(* Logix 5000 project; controller Lavado Emulate 5570 rev 32.11; software revision 32.00 *)
// Lavadora de botellas simplificada; ciclo automatico continuo basado en GRAFCET Nivel 3 v02 y CR-001; cambio CR-002.

TASK MainTask (continuous, watchdog 500 ms) : P_Lavadora

MODULES
   Local : Emulate 5570 (ICP 2, rev 32.11)
END_MODULES

VAR_GLOBAL   (* controller tags *)
   ACT_LAV_Alineacion : BOOL;   // Salida NX: 1 extiende alineador; 0 retrae.
   ACT_LAV_Banda : BOOL;   // Salida NX: 1 mueve banda; 0 detiene.
   ACT_LAV_CierrePinzas : BOOL;   // Salida NX: 1 cierra pinzas; 0 abre.
   ACT_LAV_Detencion : BOOL;   // Salida NX: 0 retiene; 1 libera.
   ACT_LAV_DetencionEntrada : BOOL;   // Salida NX CR-001: 1 extiende; 0 retrae.
   ACT_LAV_GiroLavado : BOOL;   // Salida NX: 1 gira a lavado; 0 retorna a origen.
   CMD_Inicio : BOOL;   // Pulso de inicio del automatico continuo.
   CMD_Parada : BOOL;   // Pulso de parada; cancela el lote y ordena posiciones iniciales.
   CMD_Reinicio : BOOL;   // Pulso de reinicio; borra etapas, contadores y temporizadores y ordena posiciones iniciales.
   SE_LAV_Alineado : BOOL;   // Entrada NX: alineador extendido.
   SE_LAV_CierrePinza : BOOL;   // Entrada NX: pinzas cerradas.
   SE_LAV_ConteoSalida : BOOL;   // Entrada NX: sensor de salida; cuenta por flanco ascendente.
   SE_LAV_DetencionEntradaExtendido : BOOL;   // Entrada NX CR-001: detencion de entrada extendida.
   SE_LAV_DetencionEntradaRetraido : BOOL := 1;   // Entrada NX CR-001: detencion de entrada retraida.
   SE_LAV_EntradaBotellas : BOOL;   // Entrada NX: sensor de entrada; cuenta por flanco ascendente.
   SE_LAV_Giro : BOOL;   // Entrada NX: giro en posicion de lavado.
   SE_LAV_SinAlinear : BOOL := 1;   // Entrada NX: alineador retraido.
   SE_LAV_SinDetencion : BOOL;   // Entrada NX: brazo de salida retirado y paso libre.
   SE_LAV_SinGiro : BOOL := 1;   // Entrada NX: giro en origen.
   T_Cierre : TIMER := (PRE := 1000);
END_VAR

PROGRAM P_Lavadora   (* main routine R00_Main *)
// Control secuencial simplificado; tres mandos, dos contadores, dos temporizadores y ciclo continuo.
VAR
   C_EntradaLote : COUNTER := (PRE := 7);   // Cuenta siete botellas de entrada por flanco ascendente.
   C_SalidaLote : COUNTER := (PRE := 7);   // Cuenta siete botellas de salida por flanco ascendente.
   MEM_ONS_ConteoSalida : BOOL;   // Memoria ONS exclusiva del sensor de salida.
   MEM_ONS_EntradaBotellas : BOOL;   // Memoria ONS exclusiva del sensor de entrada.
   MEM_ONS_Inicio : BOOL;   // Memoria ONS exclusiva de CMD_Inicio.
   MEM_ONS_Parada : BOOL;   // Memoria ONS exclusiva de CMD_Parada.
   MEM_ONS_Reinicio : BOOL;   // Memoria ONS exclusiva de CMD_Reinicio.
   PUL_EntradaBotella : BOOL;   // Pulso de un scan por botella de entrada.
   PUL_Inicio : BOOL;   // Pulso de un scan para inicio.
   PUL_Parada : BOOL;   // Pulso de un scan para parada.
   PUL_Reinicio : BOOL;   // Pulso de un scan para reinicio.
   PUL_SalidaBotella : BOOL;   // Pulso de un scan por botella de salida.
   ST_CicloAutomatico : BOOL;   // Memoria de marcha del ciclo automatico continuo.
   ST_LoteEntradaCompleto : BOOL;   // Memoria del septimo flanco de entrada antes del RES.
   ST_LoteSalidaCompleto : BOOL;   // Memoria del septimo flanco de salida antes del RES.
   T_Asentamiento : TIMER := (PRE := 2500);   // Ajuste de posicion de botellas despues de extender la detencion de entrada.
   T_Lavado : TIMER := (PRE := 3000);   // Tiempo de lavado del lote.
   T_Lavado_pos : TIMER := (PRE := 1000);
   TR_T00 : BOOL;   // Transicion de espera a alimentacion.
   TR_T10 : BOOL;   // Transicion despues de siete entradas.
   TR_T100 : BOOL;   // Transicion despues de siete salidas.
   TR_T105 : BOOL;   // Transicion con fin de lote seguro.
   TR_T110 : BOOL;   // Transicion automatica al siguiente lote.
   TR_T12 : BOOL;   // Transicion con detencion de entrada extendida.
   TR_T15 : BOOL;   // Transicion al completar posicionamiento.
   TR_T20 : BOOL;   // Transicion con alineador extendido.
   TR_T30 : BOOL;   // Transicion con pinzas cerradas.
   TR_T40 : BOOL;   // Transicion con giro en lavado.
   TR_T50 : BOOL;   // Transicion al completar tiempo de lavado.
   TR_T60 : BOOL;   // Transicion con giro en origen.
   TR_T70 : BOOL;   // Transicion con pinzas abiertas.
   TR_T80 : BOOL;   // Transicion con alineador retraido.
   TR_T90 : BOOL;   // Transicion con salida liberada.
   X00_Inicial : BOOL := 1;   // Etapa 0: espera de inicio y posiciones iniciales.
   X100_EvacuandoLote : BOOL;   // Etapa 100: evacuar y contar salidas.
   X105_CerrandoSalidaFinLote : BOOL;   // Etapa 105: cerrar salida y confirmar fin seguro.
   X10_Alimentando : BOOL;   // Etapa 10: alimentar y contar entradas.
   X110_RetraiendoDetencionEntrada : BOOL;   // Etapa 110: retraer detencion de entrada.
   X12_ExtendiendoDetencionEntrada : BOOL;   // Etapa 12: extender detencion de entrada con banda activa.
   X15_Posicionando : BOOL;   // Etapa 15: acomodar lote con banda activa.
   X20_Alineando : BOOL;   // Etapa 20: extender alineador.
   X30_CerrandoPinzas : BOOL;   // Etapa 30: cerrar pinzas.
   X40_GirandoLavado : BOOL;   // Etapa 40: girar hacia lavado.
   X50_Lavando : BOOL;   // Etapa 50: mantener lavado temporizado.
   X60_RegresandoGiro : BOOL;   // Etapa 60: regresar giro al origen.
   X70_AbriendoPinzas : BOOL;   // Etapa 70: abrir pinzas.
   X80_RetirandoAlineador : BOOL;   // Etapa 80: retraer alineador.
   X90_DesbloqueandoSalida : BOOL;   // Etapa 90: liberar salida.
END_VAR

ROUTINE R00_Main   (* ladder *)
// Despacha seis rutinas en orden determinista de scan.
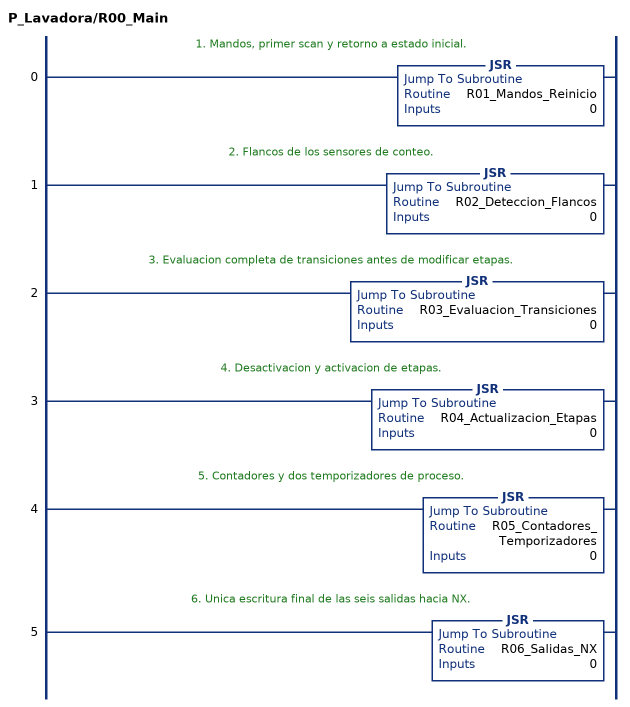
   // 1. Mandos, primer scan y retorno a estado inicial.
   0: JSR(R01_Mandos_Reinicio,0);
   // 2. Flancos de los sensores de conteo.
   1: JSR(R02_Deteccion_Flancos,0);
   // 3. Evaluacion completa de transiciones antes de modificar etapas.
   2: JSR(R03_Evaluacion_Transiciones,0);
   // 4. Desactivacion y activacion de etapas.
   3: JSR(R04_Actualizacion_Etapas,0);
   // 5. Contadores y dos temporizadores de proceso.
   4: JSR(R05_Contadores_Temporizadores,0);
   // 6. Unica escritura final de las seis salidas hacia NX.
   5: JSR(R06_Salidas_NX,0);
END_ROUTINE

ROUTINE R01_Mandos_Reinicio   (* ladder *)
// Tres mandos: inicio, parada y reinicio; parada/reinicio ordenan estado inicial.
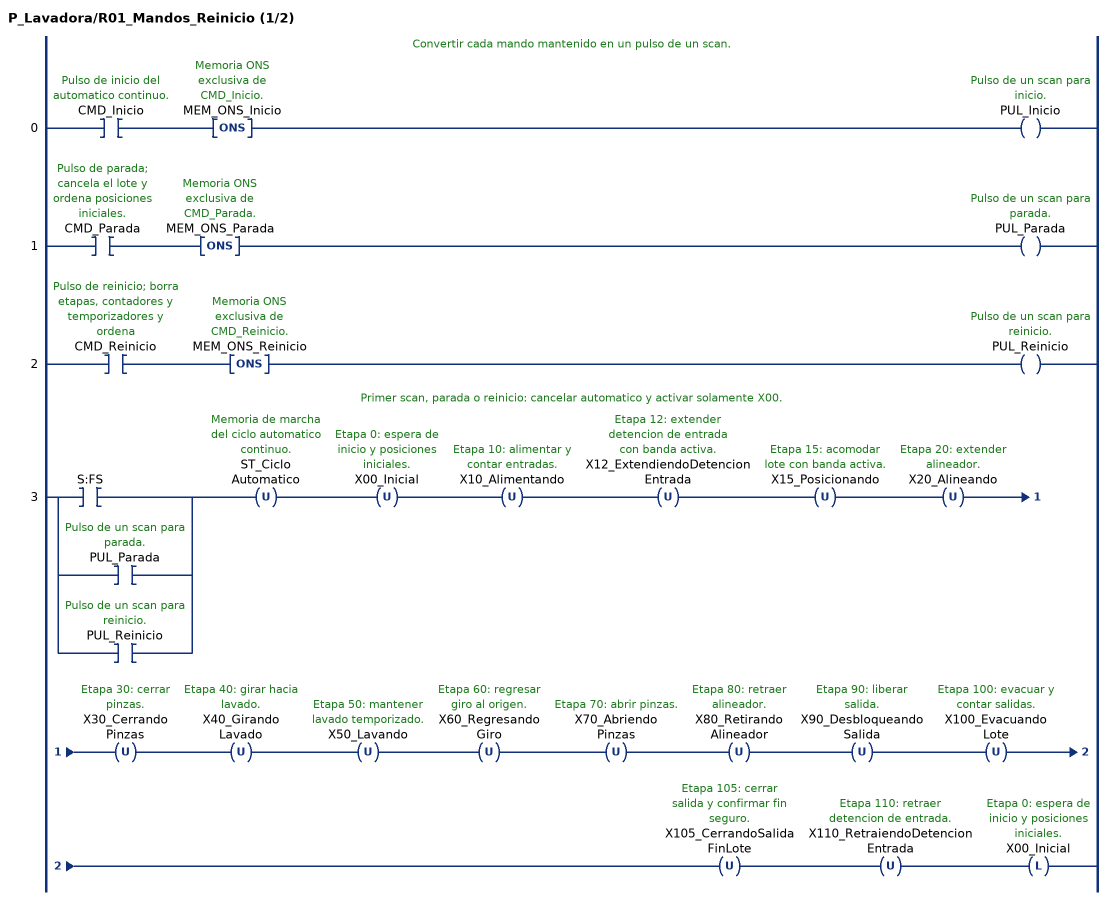
   // Convertir cada mando mantenido en un pulso de un scan.
   0: XIC(CMD_Inicio)ONS(MEM_ONS_Inicio)OTE(PUL_Inicio);
   1: XIC(CMD_Parada)ONS(MEM_ONS_Parada)OTE(PUL_Parada);
   2: XIC(CMD_Reinicio)ONS(MEM_ONS_Reinicio)OTE(PUL_Reinicio);
   // Primer scan, parada o reinicio: cancelar automatico y activar solamente X00.
   3: [XIC(S:FS) ,XIC(PUL_Parada) ,XIC(PUL_Reinicio) ]OTU(ST_CicloAutomatico)OTU(X00_Inicial)OTU(X10_Alimentando)OTU(X12_ExtendiendoDetencionEntrada)OTU(X15_Posicionando)OTU(X20_Alineando)OTU(X30_CerrandoPinzas)OTU(X40_GirandoLavado)OTU(X50_Lavando)OTU(X60_RegresandoGiro)OTU(X70_AbriendoPinzas)OTU(X80_RetirandoAlineador)OTU(X90_DesbloqueandoSalida)OTU(X100_EvacuandoLote)OTU(X105_CerrandoSalidaFinLote)OTU(X110_RetraiendoDetencionEntrada)OTL(X00_Inicial);
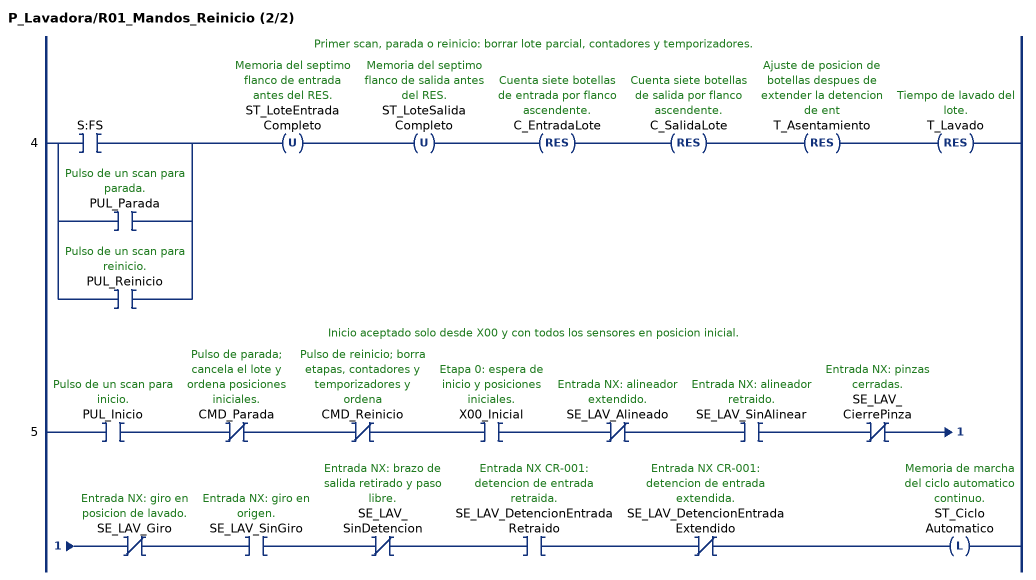
   // Primer scan, parada o reinicio: borrar lote parcial, contadores y temporizadores.
   4: [XIC(S:FS) ,XIC(PUL_Parada) ,XIC(PUL_Reinicio) ]OTU(ST_LoteEntradaCompleto)OTU(ST_LoteSalidaCompleto)RES(C_EntradaLote)RES(C_SalidaLote)RES(T_Asentamiento)RES(T_Lavado);
   // Inicio aceptado solo desde X00 y con todos los sensores en posicion inicial.
   5: XIC(PUL_Inicio)XIO(CMD_Parada)XIO(CMD_Reinicio)XIC(X00_Inicial)XIO(SE_LAV_Alineado)XIC(SE_LAV_SinAlinear)XIO(SE_LAV_CierrePinza)XIO(SE_LAV_Giro)XIC(SE_LAV_SinGiro)XIO(SE_LAV_SinDetencion)XIC(SE_LAV_DetencionEntradaRetraido)XIO(SE_LAV_DetencionEntradaExtendido)OTL(ST_CicloAutomatico);
END_ROUTINE

ROUTINE R02_Deteccion_Flancos   (* ladder *)
// Cuenta una vez cada botella aunque el sensor permanezca activo.
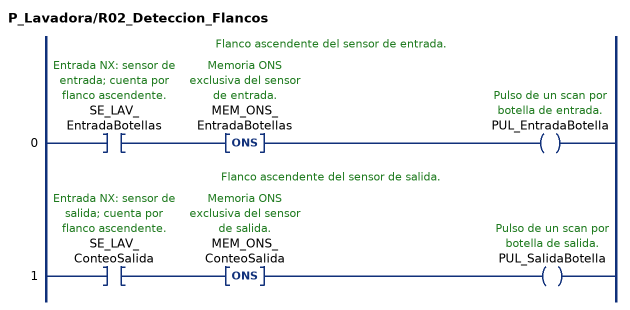
   // Flanco ascendente del sensor de entrada.
   0: XIC(SE_LAV_EntradaBotellas)ONS(MEM_ONS_EntradaBotellas)OTE(PUL_EntradaBotella);
   // Flanco ascendente del sensor de salida.
   1: XIC(SE_LAV_ConteoSalida)ONS(MEM_ONS_ConteoSalida)OTE(PUL_SalidaBotella);
END_ROUTINE

ROUTINE R03_Evaluacion_Transiciones   (* ladder *)
// Evalua las quince transiciones del GRAFCET sin modificar etapas.
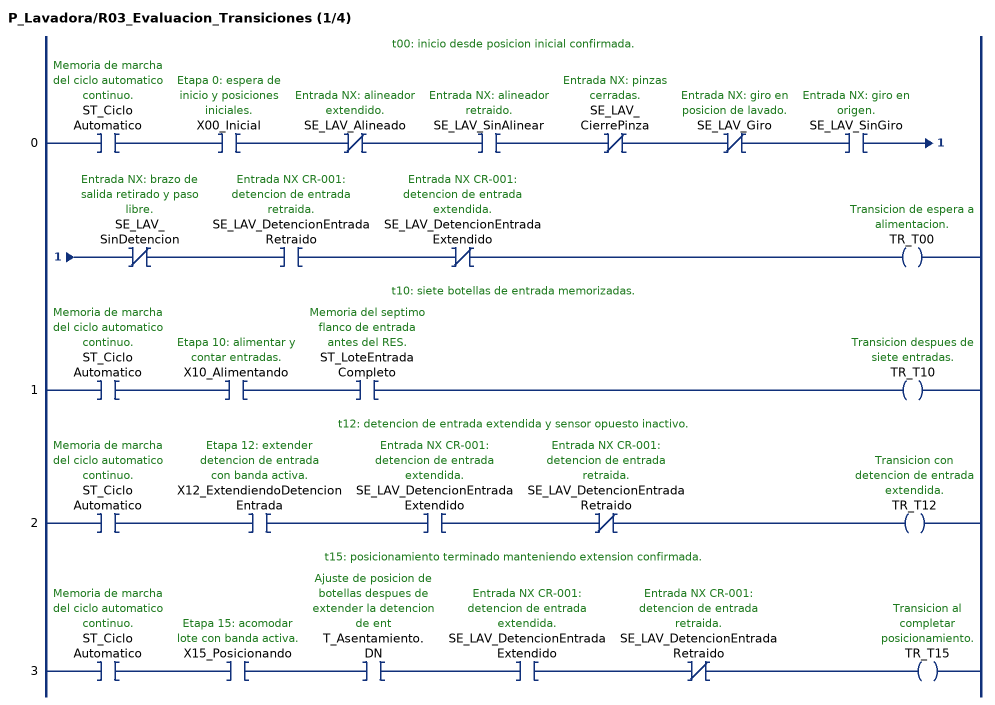
   // t00: inicio desde posicion inicial confirmada.
   0: XIC(ST_CicloAutomatico)XIC(X00_Inicial)XIO(SE_LAV_Alineado)XIC(SE_LAV_SinAlinear)XIO(SE_LAV_CierrePinza)XIO(SE_LAV_Giro)XIC(SE_LAV_SinGiro)XIO(SE_LAV_SinDetencion)XIC(SE_LAV_DetencionEntradaRetraido)XIO(SE_LAV_DetencionEntradaExtendido)OTE(TR_T00);
   // t10: siete botellas de entrada memorizadas.
   1: XIC(ST_CicloAutomatico)XIC(X10_Alimentando)XIC(ST_LoteEntradaCompleto)OTE(TR_T10);
   // t12: detencion de entrada extendida y sensor opuesto inactivo.
   2: XIC(ST_CicloAutomatico)XIC(X12_ExtendiendoDetencionEntrada)XIC(SE_LAV_DetencionEntradaExtendido)XIO(SE_LAV_DetencionEntradaRetraido)OTE(TR_T12);
   // t15: posicionamiento terminado manteniendo extension confirmada.
   3: XIC(ST_CicloAutomatico)XIC(X15_Posicionando)XIC(T_Asentamiento.DN)XIC(SE_LAV_DetencionEntradaExtendido)XIO(SE_LAV_DetencionEntradaRetraido)OTE(TR_T15);
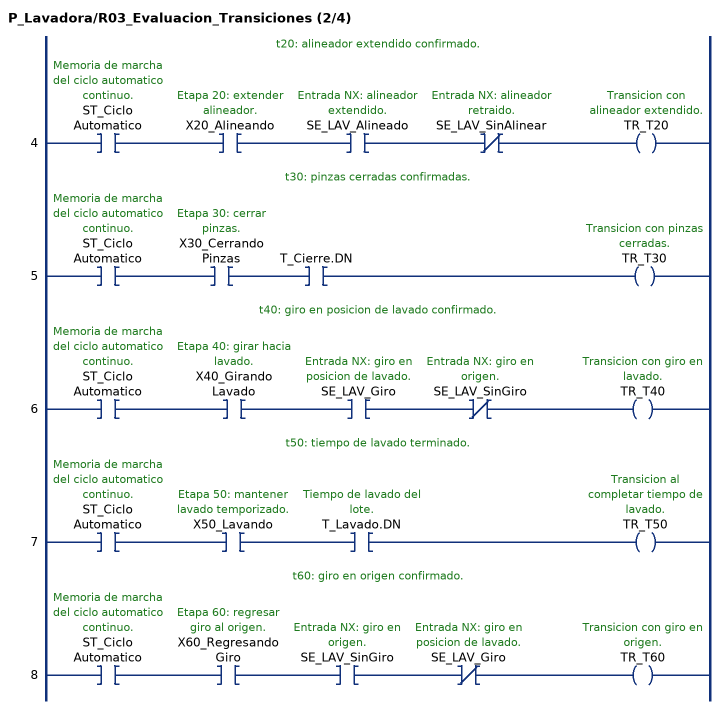
   // t20: alineador extendido confirmado.
   4: XIC(ST_CicloAutomatico)XIC(X20_Alineando)XIC(SE_LAV_Alineado)XIO(SE_LAV_SinAlinear)OTE(TR_T20);
   // t30: pinzas cerradas confirmadas.
   5: XIC(ST_CicloAutomatico)XIC(X30_CerrandoPinzas)XIC(T_Cierre.DN)OTE(TR_T30);
   // t40: giro en posicion de lavado confirmado.
   6: XIC(ST_CicloAutomatico)XIC(X40_GirandoLavado)XIC(SE_LAV_Giro)XIO(SE_LAV_SinGiro)OTE(TR_T40);
   // t50: tiempo de lavado terminado.
   7: XIC(ST_CicloAutomatico)XIC(X50_Lavando)XIC(T_Lavado.DN)OTE(TR_T50);
   // t60: giro en origen confirmado.
   8: XIC(ST_CicloAutomatico)XIC(X60_RegresandoGiro)XIC(SE_LAV_SinGiro)XIO(SE_LAV_Giro)OTE(TR_T60);
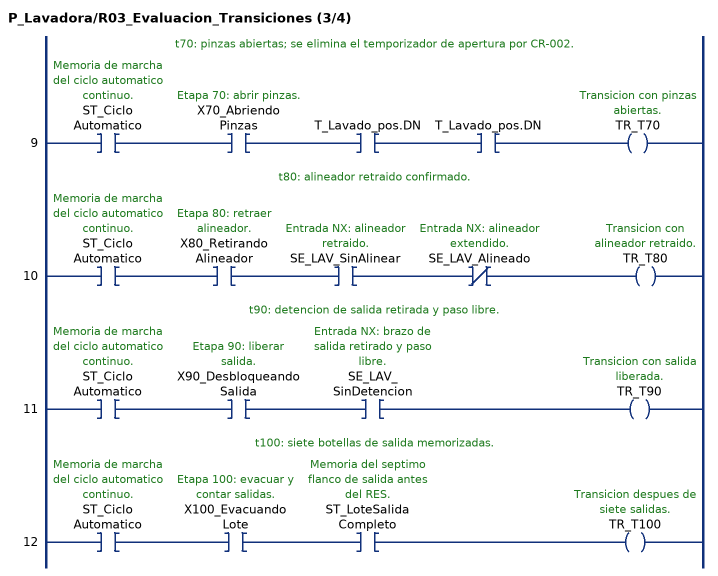
   // t70: pinzas abiertas; se elimina el temporizador de apertura por CR-002.
   9: XIC(ST_CicloAutomatico)XIC(X70_AbriendoPinzas)XIC(T_Lavado_pos.DN)XIC(T_Lavado_pos.DN)OTE(TR_T70);
   // t80: alineador retraido confirmado.
   10: XIC(ST_CicloAutomatico)XIC(X80_RetirandoAlineador)XIC(SE_LAV_SinAlinear)XIO(SE_LAV_Alineado)OTE(TR_T80);
   // t90: detencion de salida retirada y paso libre.
   11: XIC(ST_CicloAutomatico)XIC(X90_DesbloqueandoSalida)XIC(SE_LAV_SinDetencion)OTE(TR_T90);
   // t100: siete botellas de salida memorizadas.
   12: XIC(ST_CicloAutomatico)XIC(X100_EvacuandoLote)XIC(ST_LoteSalidaCompleto)OTE(TR_T100);
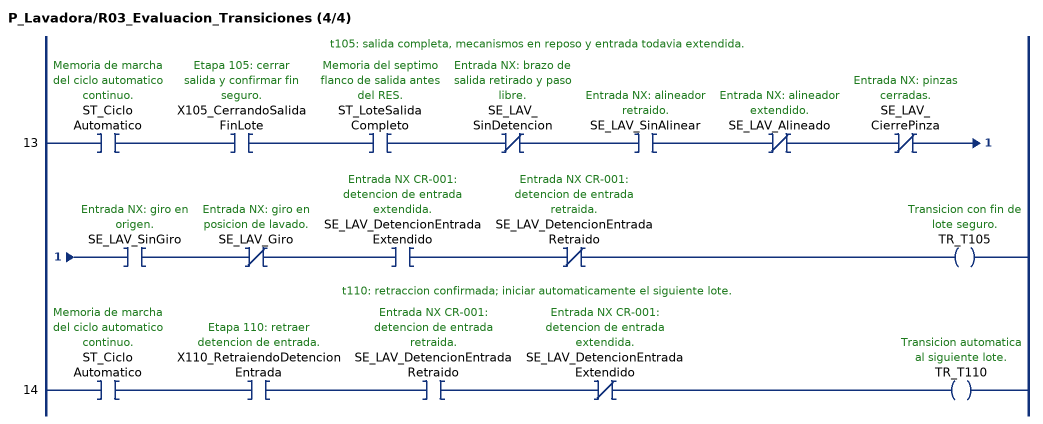
   // t105: salida completa, mecanismos en reposo y entrada todavia extendida.
   13: XIC(ST_CicloAutomatico)XIC(X105_CerrandoSalidaFinLote)XIC(ST_LoteSalidaCompleto)XIO(SE_LAV_SinDetencion)XIC(SE_LAV_SinAlinear)XIO(SE_LAV_Alineado)XIO(SE_LAV_CierrePinza)XIC(SE_LAV_SinGiro)XIO(SE_LAV_Giro)XIC(SE_LAV_DetencionEntradaExtendido)XIO(SE_LAV_DetencionEntradaRetraido)OTE(TR_T105);
   // t110: retraccion confirmada; iniciar automaticamente el siguiente lote.
   14: XIC(ST_CicloAutomatico)XIC(X110_RetraiendoDetencionEntrada)XIC(SE_LAV_DetencionEntradaRetraido)XIO(SE_LAV_DetencionEntradaExtendido)OTE(TR_T110);
END_ROUTINE

ROUTINE R04_Actualizacion_Etapas   (* ladder *)
// Aplica cada transicion evaluada: primero OTU y despues OTL.
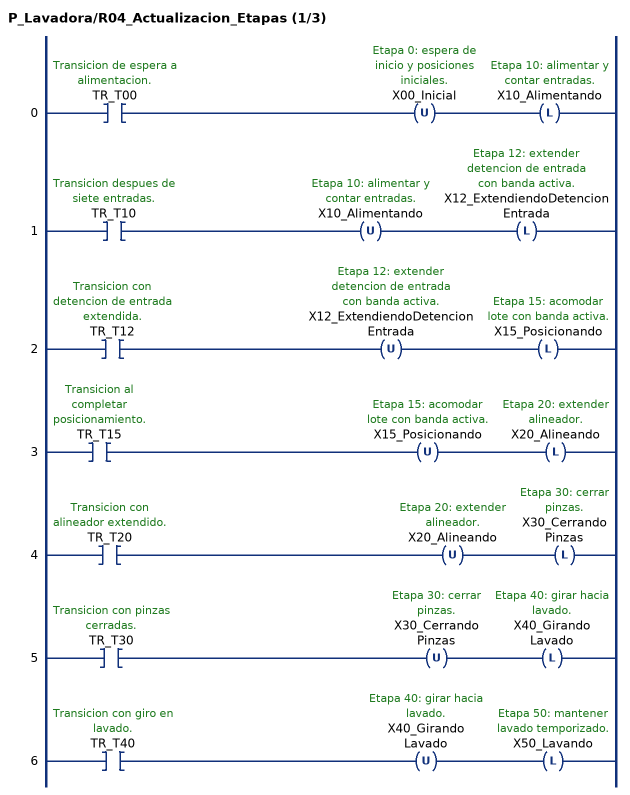
   0: XIC(TR_T00)OTU(X00_Inicial)OTL(X10_Alimentando);
   1: XIC(TR_T10)OTU(X10_Alimentando)OTL(X12_ExtendiendoDetencionEntrada);
   2: XIC(TR_T12)OTU(X12_ExtendiendoDetencionEntrada)OTL(X15_Posicionando);
   3: XIC(TR_T15)OTU(X15_Posicionando)OTL(X20_Alineando);
   4: XIC(TR_T20)OTU(X20_Alineando)OTL(X30_CerrandoPinzas);
   5: XIC(TR_T30)OTU(X30_CerrandoPinzas)OTL(X40_GirandoLavado);
   6: XIC(TR_T40)OTU(X40_GirandoLavado)OTL(X50_Lavando);
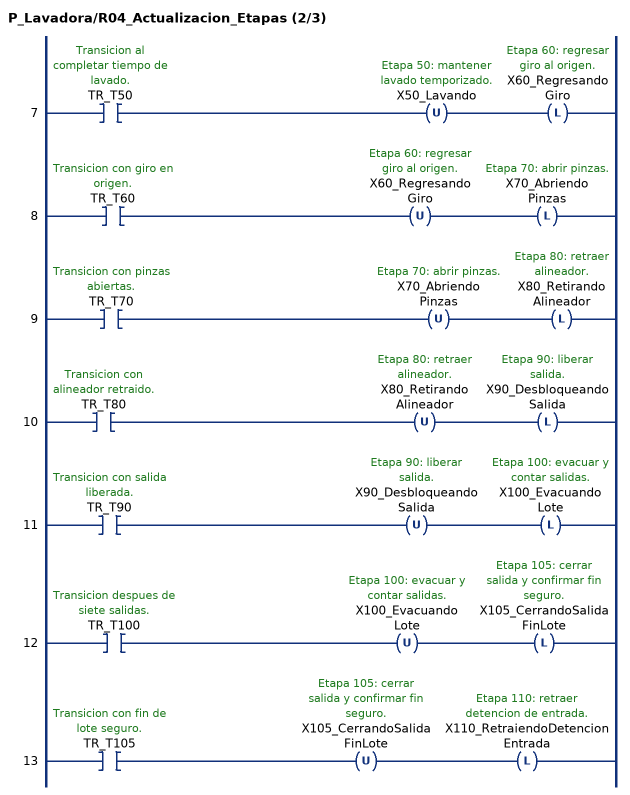
   7: XIC(TR_T50)OTU(X50_Lavando)OTL(X60_RegresandoGiro);
   8: XIC(TR_T60)OTU(X60_RegresandoGiro)OTL(X70_AbriendoPinzas);
   9: XIC(TR_T70)OTU(X70_AbriendoPinzas)OTL(X80_RetirandoAlineador);
   10: XIC(TR_T80)OTU(X80_RetirandoAlineador)OTL(X90_DesbloqueandoSalida);
   11: XIC(TR_T90)OTU(X90_DesbloqueandoSalida)OTL(X100_EvacuandoLote);
   12: XIC(TR_T100)OTU(X100_EvacuandoLote)OTL(X105_CerrandoSalidaFinLote);
   13: XIC(TR_T105)OTU(X105_CerrandoSalidaFinLote)OTL(X110_RetraiendoDetencionEntrada);
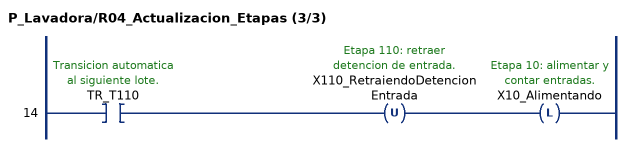
   14: XIC(TR_T110)OTU(X110_RetraiendoDetencionEntrada)OTL(X10_Alimentando);
END_ROUTINE

ROUTINE R05_Contadores_Temporizadores   (* ladder *)
// Dos CTU por flanco y dos TON de proceso; sin timeouts.
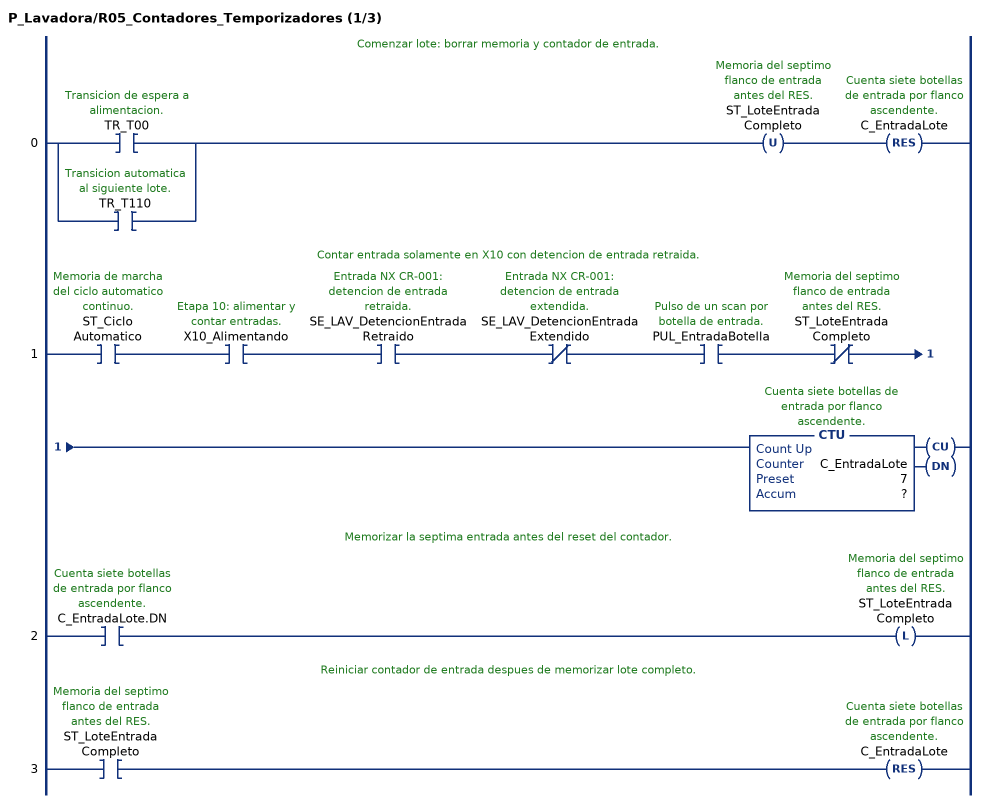
   // Comenzar lote: borrar memoria y contador de entrada.
   0: [XIC(TR_T00) ,XIC(TR_T110) ]OTU(ST_LoteEntradaCompleto)RES(C_EntradaLote);
   // Contar entrada solamente en X10 con detencion de entrada retraida.
   1: XIC(ST_CicloAutomatico)XIC(X10_Alimentando)XIC(SE_LAV_DetencionEntradaRetraido)XIO(SE_LAV_DetencionEntradaExtendido)XIC(PUL_EntradaBotella)XIO(ST_LoteEntradaCompleto)CTU(C_EntradaLote,?,?);
   // Memorizar la septima entrada antes del reset del contador.
   2: XIC(C_EntradaLote.DN)OTL(ST_LoteEntradaCompleto);
   // Reiniciar contador de entrada despues de memorizar lote completo.
   3: XIC(ST_LoteEntradaCompleto)RES(C_EntradaLote);
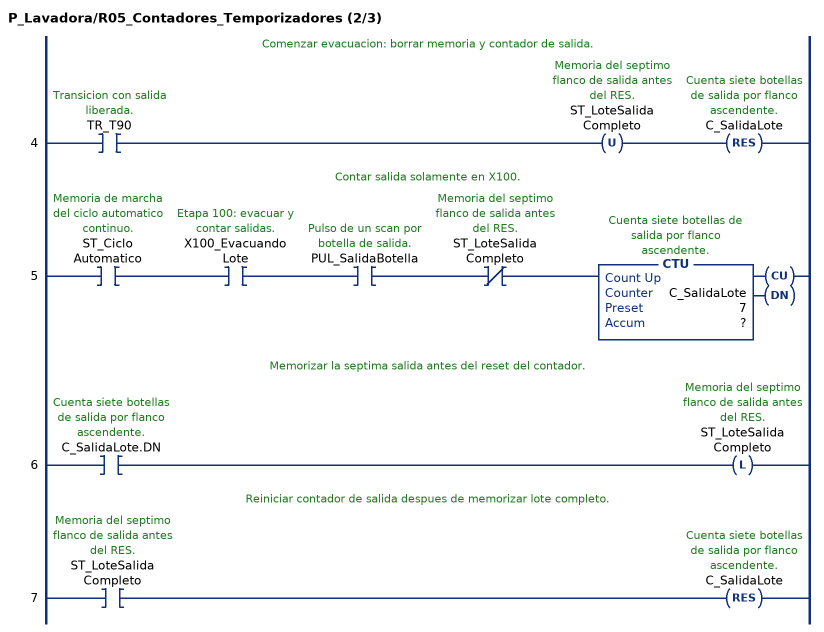
   // Comenzar evacuacion: borrar memoria y contador de salida.
   4: XIC(TR_T90)OTU(ST_LoteSalidaCompleto)RES(C_SalidaLote);
   // Contar salida solamente en X100.
   5: XIC(ST_CicloAutomatico)XIC(X100_EvacuandoLote)XIC(PUL_SalidaBotella)XIO(ST_LoteSalidaCompleto)CTU(C_SalidaLote,?,?);
   // Memorizar la septima salida antes del reset del contador.
   6: XIC(C_SalidaLote.DN)OTL(ST_LoteSalidaCompleto);
   // Reiniciar contador de salida despues de memorizar lote completo.
   7: XIC(ST_LoteSalidaCompleto)RES(C_SalidaLote);
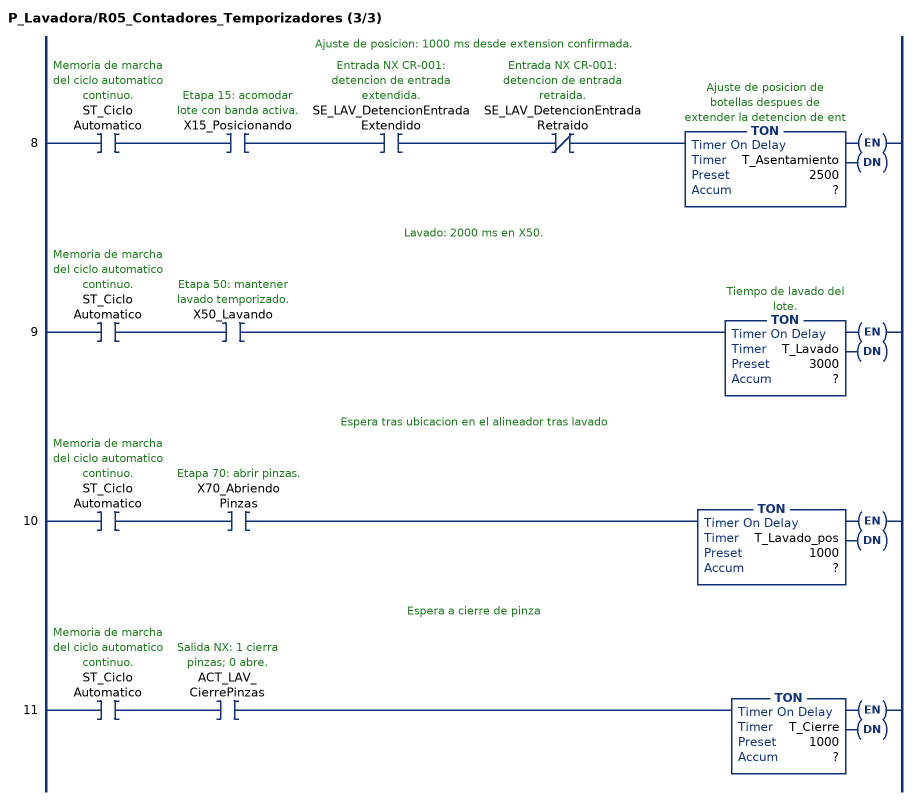
   // Ajuste de posicion: 1000 ms desde extension confirmada.
   8: XIC(ST_CicloAutomatico)XIC(X15_Posicionando)XIC(SE_LAV_DetencionEntradaExtendido)XIO(SE_LAV_DetencionEntradaRetraido)TON(T_Asentamiento,?,?);
   // Lavado: 2000 ms en X50.
   9: XIC(ST_CicloAutomatico)XIC(X50_Lavando)TON(T_Lavado,?,?);
   // Espera tras ubicacion en el alineador tras lavado
   10: XIC(ST_CicloAutomatico)XIC(X70_AbriendoPinzas)TON(T_Lavado_pos,?,?);
   // Espera a cierre de pinza
   11: XIC(ST_CicloAutomatico)XIC(ACT_LAV_CierrePinzas)TON(T_Cierre,?,?);
END_ROUTINE

ROUTINE R06_Salidas_NX   (* ladder *)
// Una unica OTE por actuador; parada o reinicio llevan todas las salidas a cero.
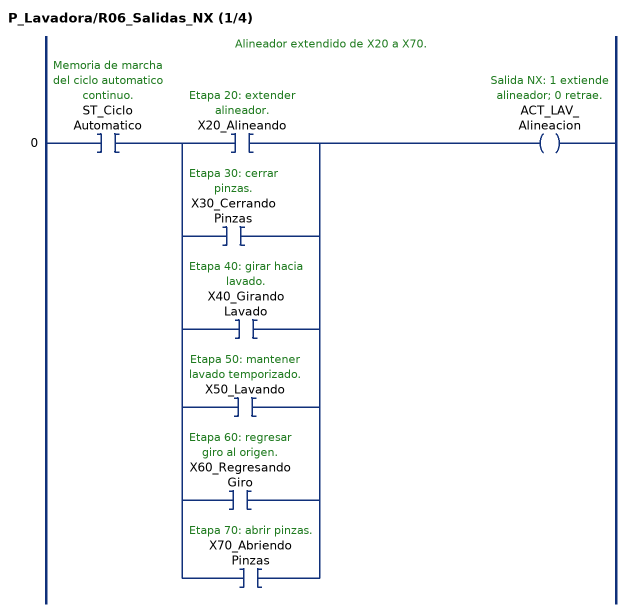
   // Alineador extendido de X20 a X70.
   0: XIC(ST_CicloAutomatico)[XIC(X20_Alineando) ,XIC(X30_CerrandoPinzas) ,XIC(X40_GirandoLavado) ,XIC(X50_Lavando) ,XIC(X60_RegresandoGiro) ,XIC(X70_AbriendoPinzas) ]OTE(ACT_LAV_Alineacion);
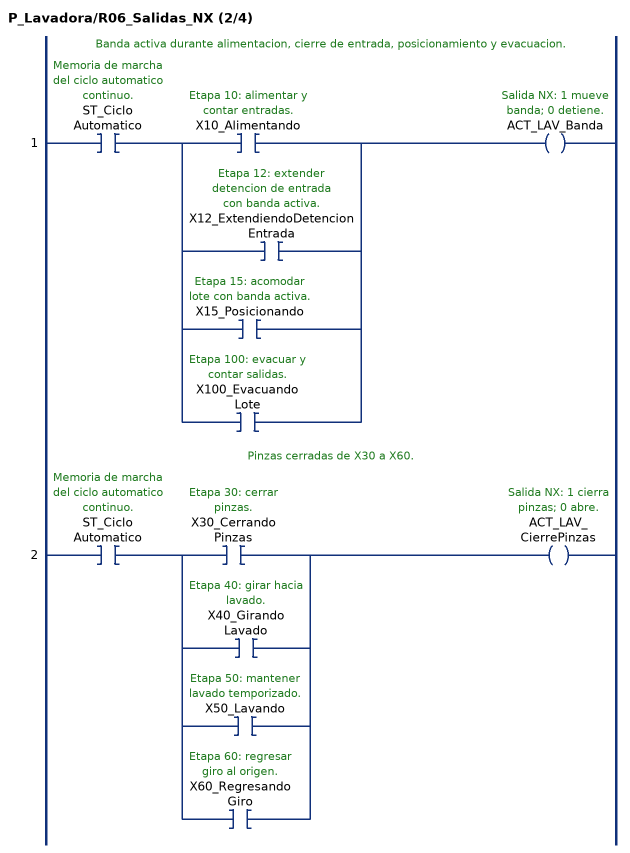
   // Banda activa durante alimentacion, cierre de entrada, posicionamiento y evacuacion.
   1: XIC(ST_CicloAutomatico)[XIC(X10_Alimentando) ,XIC(X12_ExtendiendoDetencionEntrada) ,XIC(X15_Posicionando) ,XIC(X100_EvacuandoLote) ]OTE(ACT_LAV_Banda);
   // Pinzas cerradas de X30 a X60.
   2: XIC(ST_CicloAutomatico)[XIC(X30_CerrandoPinzas) ,XIC(X40_GirandoLavado) ,XIC(X50_Lavando) ,XIC(X60_RegresandoGiro) ]OTE(ACT_LAV_CierrePinzas);
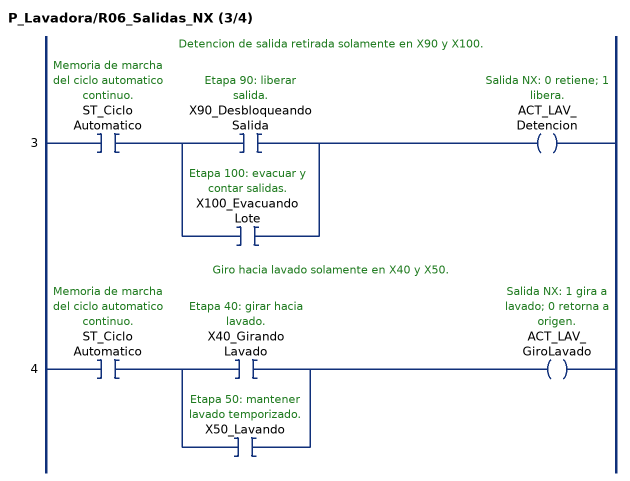
   // Detencion de salida retirada solamente en X90 y X100.
   3: XIC(ST_CicloAutomatico)[XIC(X90_DesbloqueandoSalida) ,XIC(X100_EvacuandoLote) ]OTE(ACT_LAV_Detencion);
   // Giro hacia lavado solamente en X40 y X50.
   4: XIC(ST_CicloAutomatico)[XIC(X40_GirandoLavado) ,XIC(X50_Lavando) ]OTE(ACT_LAV_GiroLavado);
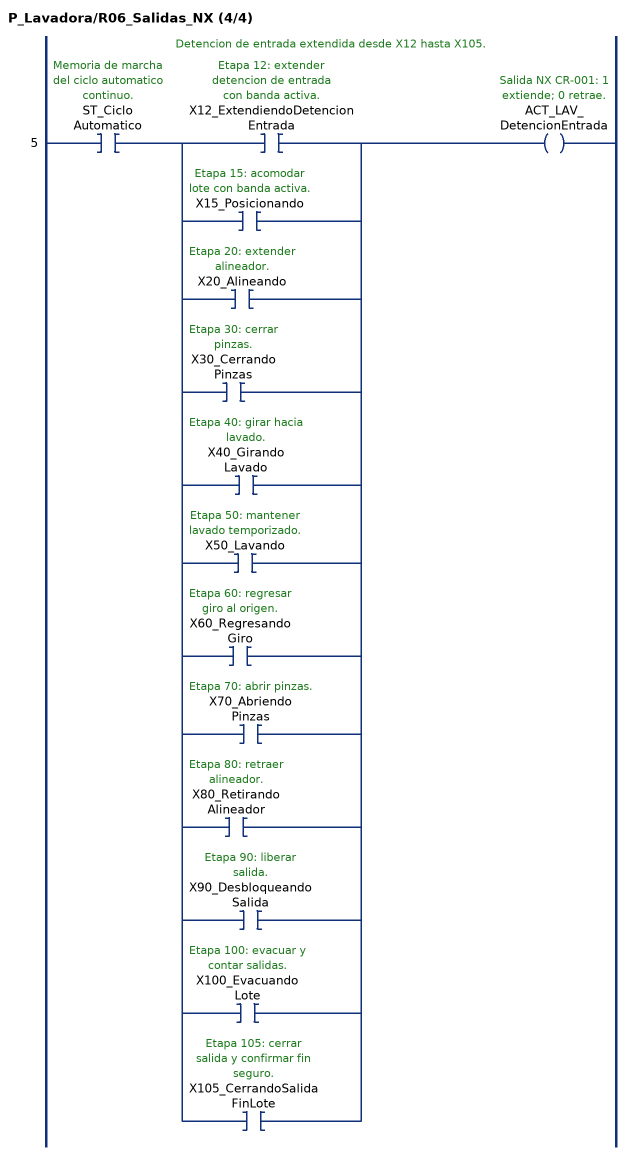
   // Detencion de entrada extendida desde X12 hasta X105.
   5: XIC(ST_CicloAutomatico)[XIC(X12_ExtendiendoDetencionEntrada) ,XIC(X15_Posicionando) ,XIC(X20_Alineando) ,XIC(X30_CerrandoPinzas) ,XIC(X40_GirandoLavado) ,XIC(X50_Lavando) ,XIC(X60_RegresandoGiro) ,XIC(X70_AbriendoPinzas) ,XIC(X80_RetirandoAlineador) ,XIC(X90_DesbloqueandoSalida) ,XIC(X100_EvacuandoLote) ,XIC(X105_CerrandoSalidaFinLote) ]OTE(ACT_LAV_DetencionEntrada);
END_ROUTINE
END_PROGRAM
